// SIMATIC S7-200 project (STEP 7-Micro/WIN), CPU 221 REL 01.10

SYMBOL_TABLE USER1
ONN              I0.0     // NHAN CHAY
OFF              I0.1     // NHAN DUNG
RESET            I0.2     // RESET TMER TONR
DC1              Q0.0
XANH             Q0.1     // DEN BAO CHAY
DO               Q0.2     // DEN BAO DUNG
VANG             Q0.3     // DEN BAO SU CO
END_SYMBOL_TABLE

ORGANIZATION_BLOCK MAIN:OB1
TITLE=PROGRAM COMMENTS
BEGIN
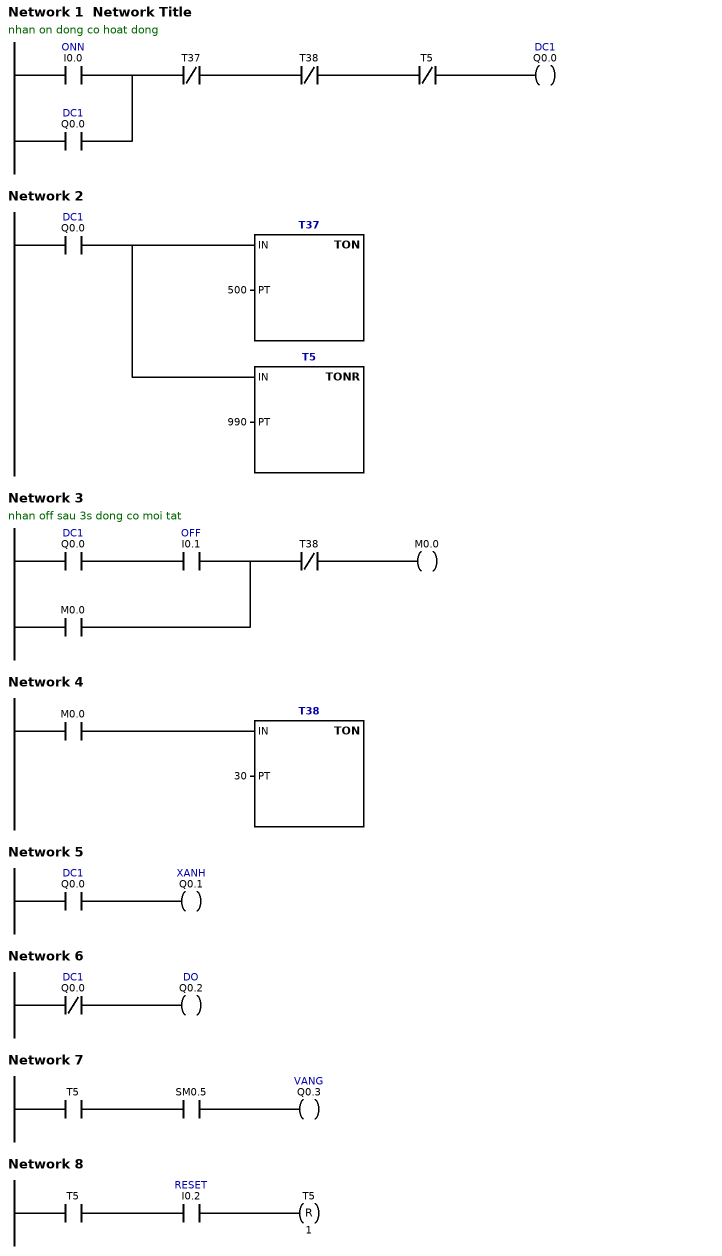
Network 1 // Network Title
// nhan on dong co hoat dong
// (network saved uncompiled; LAD cells follow)
// row 0: c0 -| |- ONN:I0.0 v  c1 -|/|- T37  c2 -|/|- T38  c3 -|/|- T5  c4 -( ) DC1:Q0.0
// row 1: c0 -| |- DC1:Q0.0 ^
Network 2
LD     DC1:Q0.0
TON    T37, 500
TONR   T5, 990
Network 3
// nhan off sau 3s dong co moi tat
LD     DC1:Q0.0
A      OFF:I0.1
O      M0.0
AN     T38
=      M0.0
Network 4
// (network saved uncompiled; LAD cells follow)
// row 0: c0 -| |- M0.0  c1 --  c2 [TON T38 IN:=power@row0, PT:=30]
// row 1: c2 [box]
Network 5
LD     DC1:Q0.0
=      XANH:Q0.1
Network 6
LDN    DC1:Q0.0
=      DO:Q0.2
Network 7
LD     T5
A      SM0.5
=      VANG:Q0.3
Network 8
LD     T5
A      RESET:I0.2
R      T5, 1
END_ORGANIZATION_BLOCK
